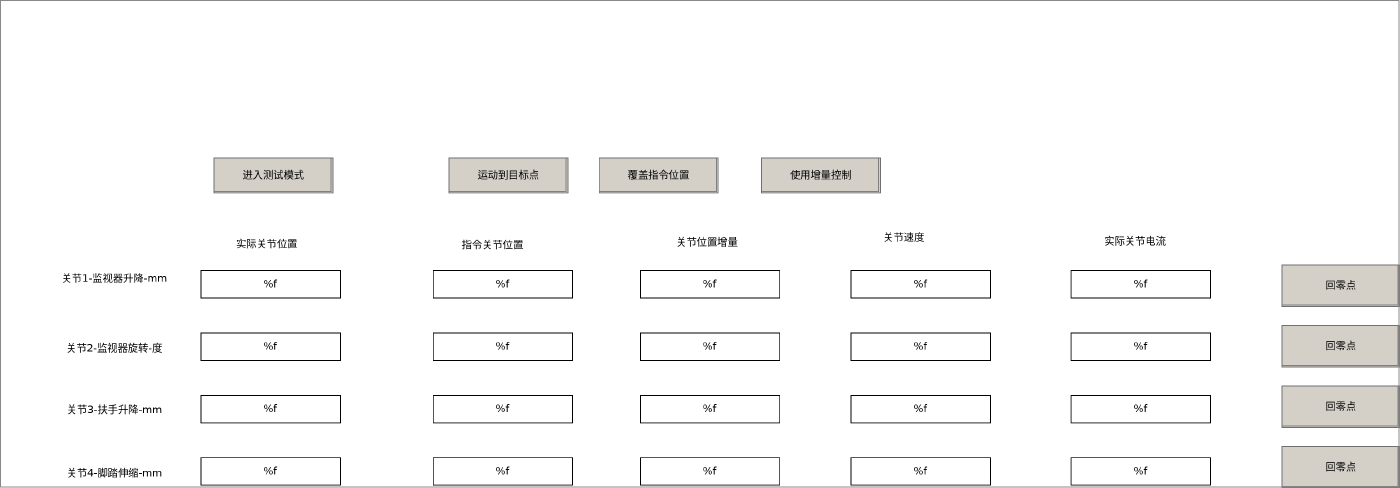
VISUALIZATION motion_car  // 1501x524
    Label (211,247 150x30), "实际关节位置"
    Rectangle (215,290 150x30), "%f", text variable: g_motionTest.m_carJntPos[1]
    Label (453,248 150x30), "指令关节位置"
    Label (683,245 150x30), "关节位置增量"
    Rectangle (686,290 150x30), "%f", text variable: g_motionTest.m_targetJntPosIncCar[1]
        OnMouseClick: write the text variable via Default
    Label (1142,244 150x30), "实际关节电流"
    Rectangle (1148,290 150x30), "%f", text variable: g_motionTest.m_carJntCurrent[1]
    Rectangle (215,357 150x30), "%f", text variable: g_motionTest.m_carJntPos[2]
    Rectangle (215,424 150x30), "%f", text variable: g_motionTest.m_carJntPos[3]
    Rectangle (215,491 150x30), "%f", text variable: g_motionTest.m_carJntPos[4]
    Rectangle (464,290 150x30), "%f", text variable: g_motionTest.m_targetJntPosCar[1]
        OnMouseClick: write the text variable via Default
    Rectangle (464,357 150x30), "%f", text variable: g_motionTest.m_targetJntPosCar[2]
        OnMouseClick: write the text variable via Default
    Rectangle (464,424 150x30), "%f", text variable: g_motionTest.m_targetJntPosCar[3]
        OnMouseClick: write the text variable via Default
    Rectangle (464,491 150x30), "%f", text variable: g_motionTest.m_targetJntPosCar[4]
        OnMouseClick: write the text variable via Default
    Rectangle (686,357 150x30), "%f", text variable: g_motionTest.m_targetJntPosIncCar[2]
        OnMouseClick: write the text variable via Default
    Rectangle (686,424 150x30), "%f", text variable: g_motionTest.m_targetJntPosIncCar[3]
        OnMouseClick: write the text variable via Default
    Rectangle (686,491 150x30), "%f", text variable: g_motionTest.m_targetJntPosIncCar[4]
        OnMouseClick: write the text variable via Default
    Rectangle (1148,357 150x30), "%f", text variable: g_motionTest.m_carJntCurrent[2]
    Rectangle (1148,424 150x30), "%f", text variable: g_motionTest.m_carJntCurrent[3]
    Rectangle (1148,491 150x30), "%f", text variable: g_motionTest.m_carJntCurrent[4]
    Label (894,240 150x30), "关节速度"
    Rectangle (912,290 150x30), "%f", text variable: g_motionTest.m_targetJntVelCar[1]
        OnMouseClick: write the text variable via Default
    Rectangle (912,357 150x30), "%f", text variable: g_motionTest.m_targetJntVelCar[2]
        OnMouseClick: write the text variable via Default
    Rectangle (912,424 150x30), "%f", text variable: g_motionTest.m_targetJntVelCar[3]
        OnMouseClick: write the text variable via Default
    Rectangle (912,491 150x30), "%f", text variable: g_motionTest.m_targetJntVelCar[4]
        OnMouseClick: write the text variable via Default
    Button (229,169 128x38), "进入测试模式", colour toggle: g_motionTest.m_enterJntTestCar
        toggle g_motionTest.m_enterJntTestCar
    Button (481,169 128x38), "运动到目标点", colour toggle: g_motionTest.m_startMotionCar
        tap g_motionTest.m_startMotionCar
    Button (816,169 128x38), "使用增量控制", colour toggle: g_motionTest.m_jntPosIncModeCar
        toggle g_motionTest.m_jntPosIncModeCar
    Button (642,169 128x38), "覆盖指令位置", colour toggle: g_motionTest.m_coverCmdPosCar
        tap g_motionTest.m_coverCmdPosCar
    Label (50,285 145x28), "关节1-监视器升降-mm"
    Label (50,360 145x28), "关节2-监视器旋转-度"
    Label (50,426 145x28), "关节3-扶手升降-mm"
    Label (50,494 145x28), "关节4-脚踏伸缩-mm"
    Button (1374,284 127x45), "回零点", colour toggle: g_motionTest.m_goHomeCar[1]
        tap g_motionTest.m_goHomeCar[1]
    Button (1374,349 127x45), "回零点", colour toggle: g_motionTest.m_goHomeCar[2]
        tap g_motionTest.m_goHomeCar[2]
    Button (1374,414 127x45), "回零点", colour toggle: g_motionTest.m_goHomeCar[3]
        tap g_motionTest.m_goHomeCar[3]
    Button (1374,479 127x45), "回零点", colour toggle: g_motionTest.m_goHomeCar[4]
        tap g_motionTest.m_goHomeCar[4]
END_VISUALIZATION

(* stored: Version 1.1.0.1, ProductVersion 3.1.4024.11
   Visu motion_car: Id {14495e51-3bf5-4dc1-bb92-466eb6086a2c} *)
